# EPICS substitutions: apps/xpsMotorApp/Db/XPS2_Aux_ai.substitutions
file "db/XPSAuxAi.db"
{
pattern
{P,          R,          PORT,     CHAN, LOPR,   HOPR,  PREC, SCAN}
{halldxps2:, XPSAuxAi0,  XPS_AUX1, 0,    -10.0,  10.0,  6,    "1 second"}
{halldxps2:, XPSAuxAi1,  XPS_AUX1, 1,    -10.0,  10.0,  6,    "1 second"}
{halldxps2:, XPSAuxAi2,  XPS_AUX1, 2,    -10.0,  10.0,  6,    "1 second"}
{halldxps2:, XPSAuxAi3,  XPS_AUX1, 3,    -10.0,  10.0,  6,    "1 second"}
}
